(* Logix 5000 project; controller SX_V040001_C001 vendor 1 type 14 code 77 rev 16.22; software revision 16.04; part 26 of 35 *)
(* tags used below, declared in another part *)
   ALL_KINDS : INT[90];
   METERING : INT[44];
   PARAMETER : INT[501];
(* MainProgram, continued *)

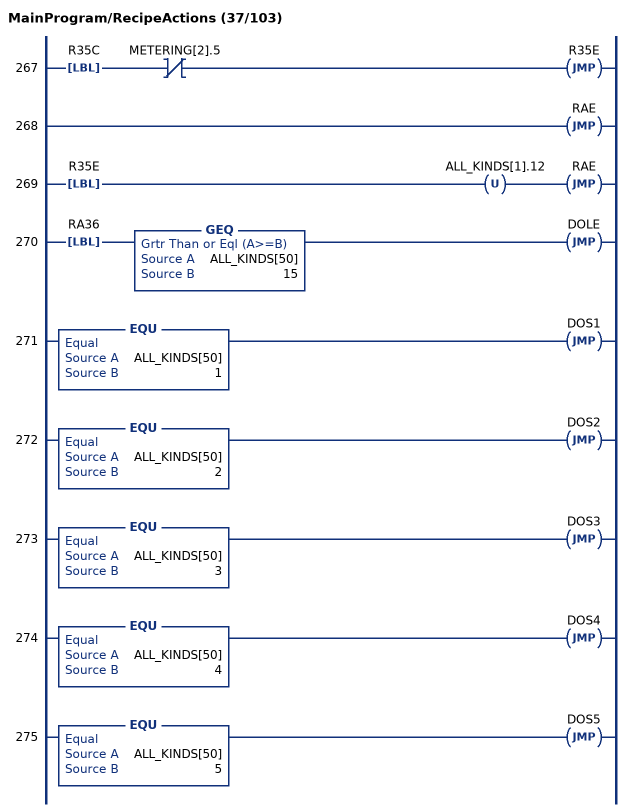
   [picture p568: MainProgram/RecipeActions rungs 267-275]
   267: LBL(R35C)XIO(METERING[2].5)JMP(R35E);
   268: JMP(RAE);
   269: LBL(R35E)OTU(ALL_KINDS[1].12)JMP(RAE);
   270: LBL(RA36)GEQ(ALL_KINDS[50],15)JMP(DOLE);
   271: EQU(ALL_KINDS[50],1)JMP(DOS1);
   272: EQU(ALL_KINDS[50],2)JMP(DOS2);
   273: EQU(ALL_KINDS[50],3)JMP(DOS3);
   274: EQU(ALL_KINDS[50],4)JMP(DOS4);
   275: EQU(ALL_KINDS[50],5)JMP(DOS5);
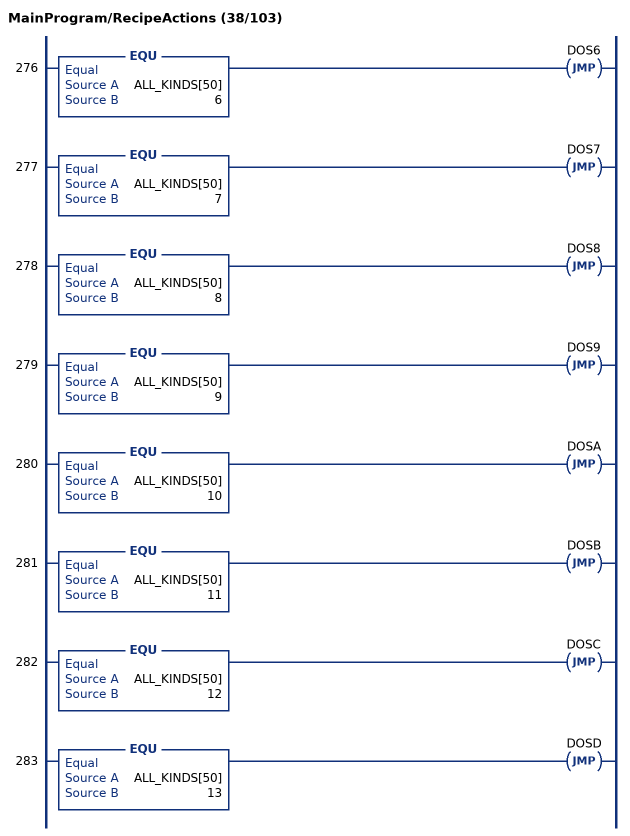
   276: EQU(ALL_KINDS[50],6)JMP(DOS6);
   277: EQU(ALL_KINDS[50],7)JMP(DOS7);
   278: EQU(ALL_KINDS[50],8)JMP(DOS8);
   279: EQU(ALL_KINDS[50],9)JMP(DOS9);
   280: EQU(ALL_KINDS[50],10)JMP(DOSA);
   281: EQU(ALL_KINDS[50],11)JMP(DOSB);
   282: EQU(ALL_KINDS[50],12)JMP(DOSC);
   283: EQU(ALL_KINDS[50],13)JMP(DOSD);
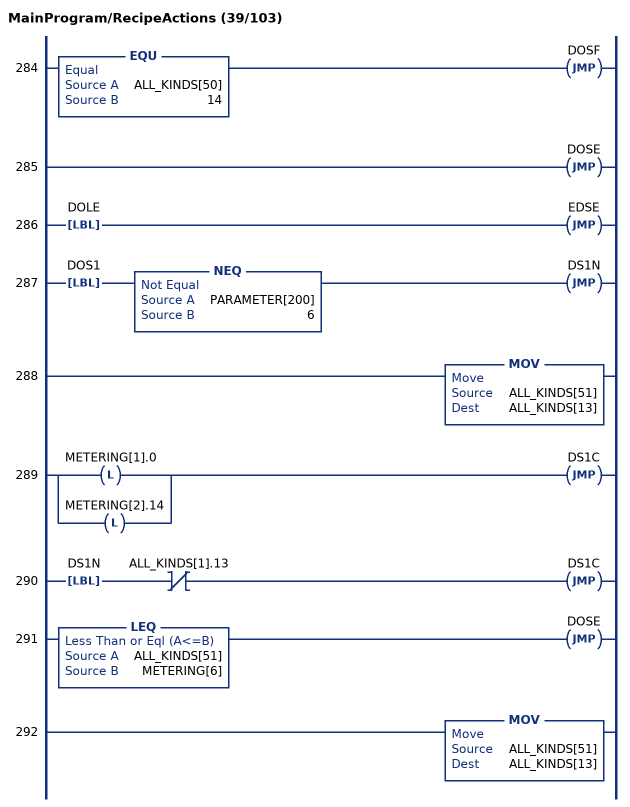
   284: EQU(ALL_KINDS[50],14)JMP(DOSF);
   285: JMP(DOSE);
   286: LBL(DOLE)JMP(EDSE);
   287: LBL(DOS1)NEQ(PARAMETER[200],6)JMP(DS1N);
   288: MOV(ALL_KINDS[51],ALL_KINDS[13]);
   289: [OTL(METERING[1].0) ,OTL(METERING[2].14) ]JMP(DS1C);
   290: LBL(DS1N)XIO(ALL_KINDS[1].13)JMP(DS1C);
   291: LEQ(ALL_KINDS[51],METERING[6])JMP(DOSE);
   292: MOV(ALL_KINDS[51],ALL_KINDS[13]);
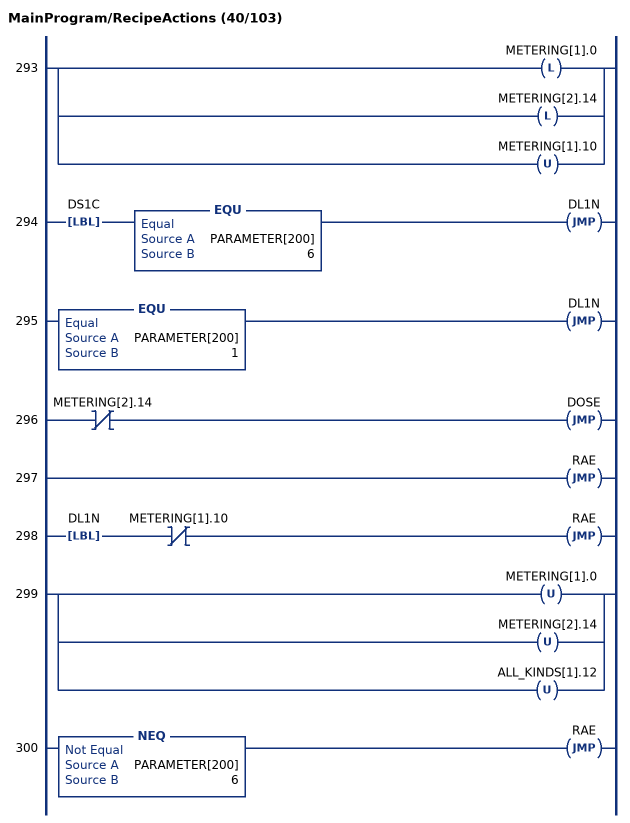
   293: [OTL(METERING[1].0) ,OTL(METERING[2].14) ,OTU(METERING[1].10) ];
   294: LBL(DS1C)EQU(PARAMETER[200],6)JMP(DL1N);
   295: EQU(PARAMETER[200],1)JMP(DL1N);
   296: XIO(METERING[2].14)JMP(DOSE);
   297: JMP(RAE);
   298: LBL(DL1N)XIO(METERING[1].10)JMP(RAE);
   299: [OTU(METERING[1].0) ,OTU(METERING[2].14) ,OTU(ALL_KINDS[1].12) ];
   300: NEQ(PARAMETER[200],6)JMP(RAE);
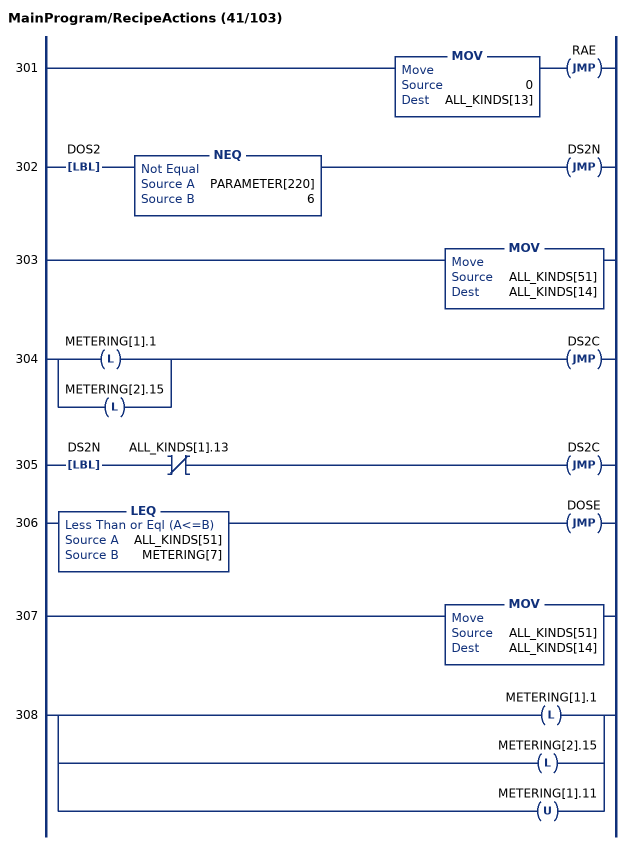
   301: MOV(0,ALL_KINDS[13])JMP(RAE);
   302: LBL(DOS2)NEQ(PARAMETER[220],6)JMP(DS2N);
   303: MOV(ALL_KINDS[51],ALL_KINDS[14]);
   304: [OTL(METERING[1].1) ,OTL(METERING[2].15) ]JMP(DS2C);
   305: LBL(DS2N)XIO(ALL_KINDS[1].13)JMP(DS2C);
   306: LEQ(ALL_KINDS[51],METERING[7])JMP(DOSE);
   307: MOV(ALL_KINDS[51],ALL_KINDS[14]);
   308: [OTL(METERING[1].1) ,OTL(METERING[2].15) ,OTU(METERING[1].11) ];
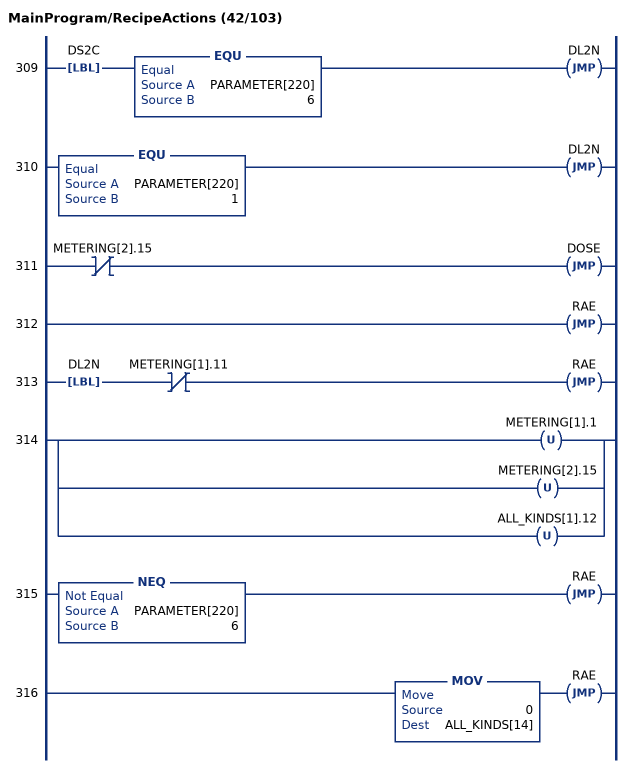
   309: LBL(DS2C)EQU(PARAMETER[220],6)JMP(DL2N);
   310: EQU(PARAMETER[220],1)JMP(DL2N);
   311: XIO(METERING[2].15)JMP(DOSE);
   312: JMP(RAE);
   313: LBL(DL2N)XIO(METERING[1].11)JMP(RAE);
   314: [OTU(METERING[1].1) ,OTU(METERING[2].15) ,OTU(ALL_KINDS[1].12) ];
   315: NEQ(PARAMETER[220],6)JMP(RAE);
   316: MOV(0,ALL_KINDS[14])JMP(RAE);
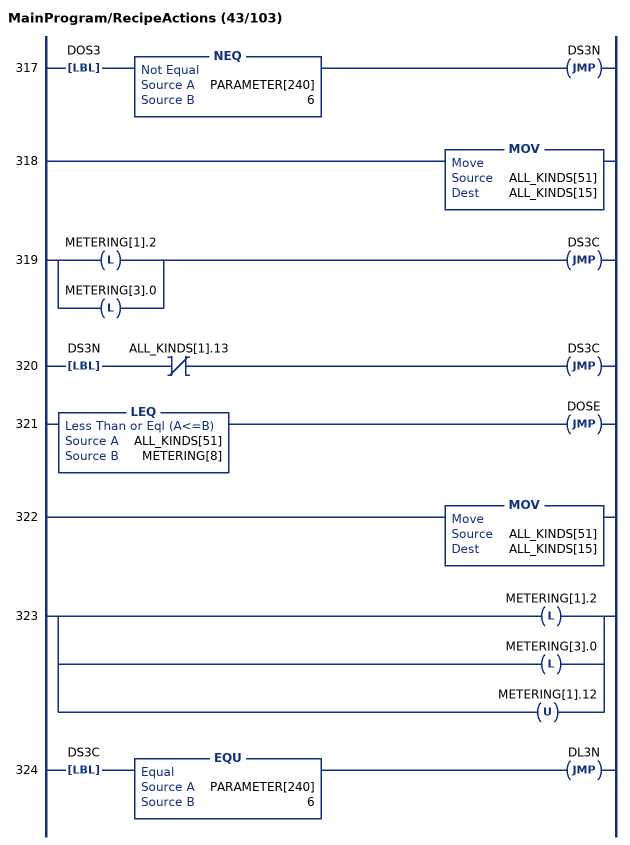
   317: LBL(DOS3)NEQ(PARAMETER[240],6)JMP(DS3N);
   318: MOV(ALL_KINDS[51],ALL_KINDS[15]);
   319: [OTL(METERING[1].2) ,OTL(METERING[3].0) ]JMP(DS3C);
   320: LBL(DS3N)XIO(ALL_KINDS[1].13)JMP(DS3C);
   321: LEQ(ALL_KINDS[51],METERING[8])JMP(DOSE);
   322: MOV(ALL_KINDS[51],ALL_KINDS[15]);
   323: [OTL(METERING[1].2) ,OTL(METERING[3].0) ,OTU(METERING[1].12) ];
   324: LBL(DS3C)EQU(PARAMETER[240],6)JMP(DL3N);
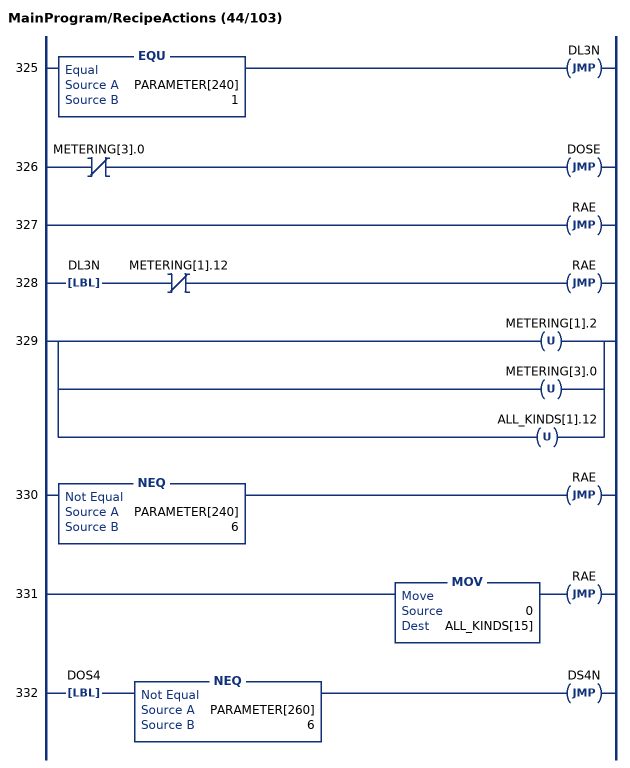
   325: EQU(PARAMETER[240],1)JMP(DL3N);
   326: XIO(METERING[3].0)JMP(DOSE);
   327: JMP(RAE);
   328: LBL(DL3N)XIO(METERING[1].12)JMP(RAE);
   329: [OTU(METERING[1].2) ,OTU(METERING[3].0) ,OTU(ALL_KINDS[1].12) ];
   330: NEQ(PARAMETER[240],6)JMP(RAE);
   331: MOV(0,ALL_KINDS[15])JMP(RAE);
   332: LBL(DOS4)NEQ(PARAMETER[260],6)JMP(DS4N);
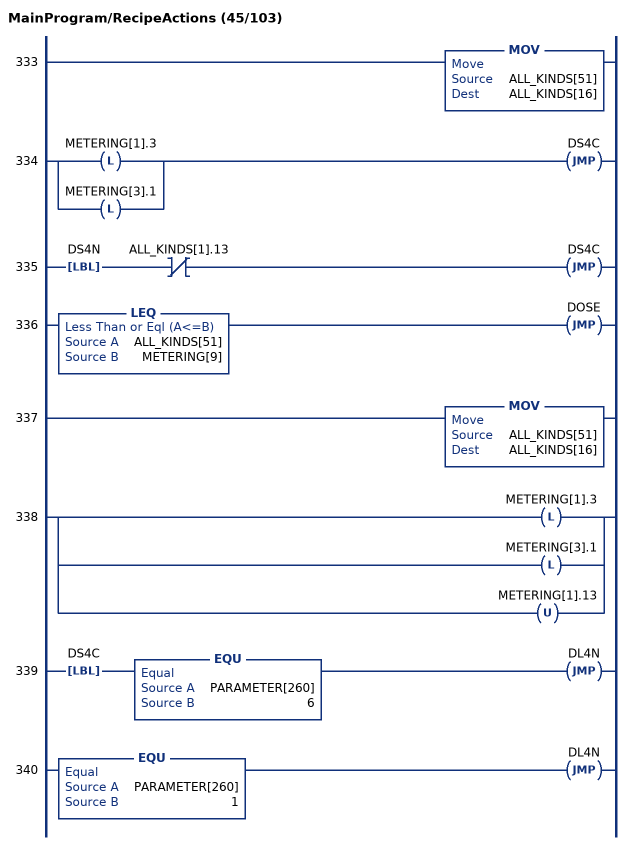
   333: MOV(ALL_KINDS[51],ALL_KINDS[16]);
   334: [OTL(METERING[1].3) ,OTL(METERING[3].1) ]JMP(DS4C);
   335: LBL(DS4N)XIO(ALL_KINDS[1].13)JMP(DS4C);
   336: LEQ(ALL_KINDS[51],METERING[9])JMP(DOSE);
   337: MOV(ALL_KINDS[51],ALL_KINDS[16]);
   338: [OTL(METERING[1].3) ,OTL(METERING[3].1) ,OTU(METERING[1].13) ];
   339: LBL(DS4C)EQU(PARAMETER[260],6)JMP(DL4N);
   340: EQU(PARAMETER[260],1)JMP(DL4N);
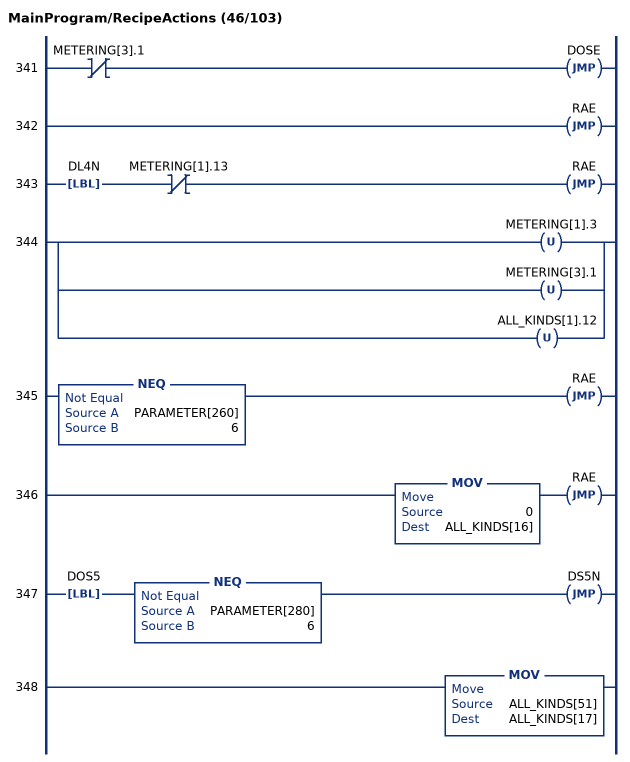
   341: XIO(METERING[3].1)JMP(DOSE);
   342: JMP(RAE);
   343: LBL(DL4N)XIO(METERING[1].13)JMP(RAE);
   344: [OTU(METERING[1].3) ,OTU(METERING[3].1) ,OTU(ALL_KINDS[1].12) ];
   345: NEQ(PARAMETER[260],6)JMP(RAE);
   346: MOV(0,ALL_KINDS[16])JMP(RAE);
   347: LBL(DOS5)NEQ(PARAMETER[280],6)JMP(DS5N);
   348: MOV(ALL_KINDS[51],ALL_KINDS[17]);
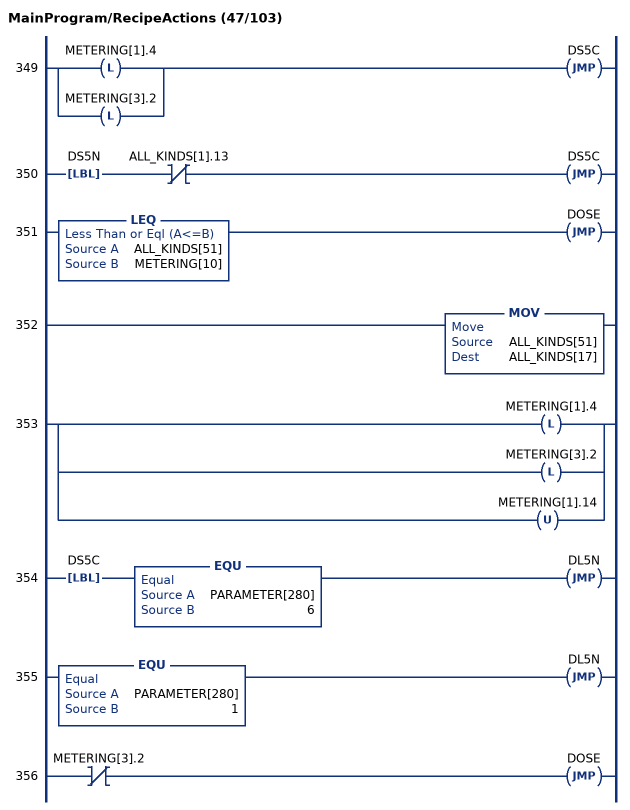
   349: [OTL(METERING[1].4) ,OTL(METERING[3].2) ]JMP(DS5C);
   350: LBL(DS5N)XIO(ALL_KINDS[1].13)JMP(DS5C);
   351: LEQ(ALL_KINDS[51],METERING[10])JMP(DOSE);
   352: MOV(ALL_KINDS[51],ALL_KINDS[17]);
   353: [OTL(METERING[1].4) ,OTL(METERING[3].2) ,OTU(METERING[1].14) ];
   354: LBL(DS5C)EQU(PARAMETER[280],6)JMP(DL5N);
   355: EQU(PARAMETER[280],1)JMP(DL5N);
   356: XIO(METERING[3].2)JMP(DOSE);
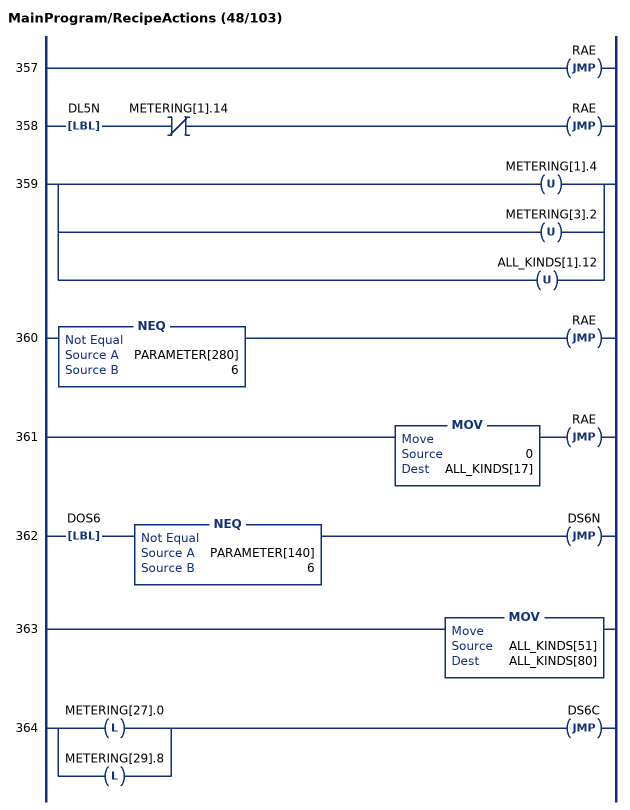
   357: JMP(RAE);
   358: LBL(DL5N)XIO(METERING[1].14)JMP(RAE);
   359: [OTU(METERING[1].4) ,OTU(METERING[3].2) ,OTU(ALL_KINDS[1].12) ];
   360: NEQ(PARAMETER[280],6)JMP(RAE);
   361: MOV(0,ALL_KINDS[17])JMP(RAE);
   362: LBL(DOS6)NEQ(PARAMETER[140],6)JMP(DS6N);
   363: MOV(ALL_KINDS[51],ALL_KINDS[80]);
   364: [OTL(METERING[27].0) ,OTL(METERING[29].8) ]JMP(DS6C);
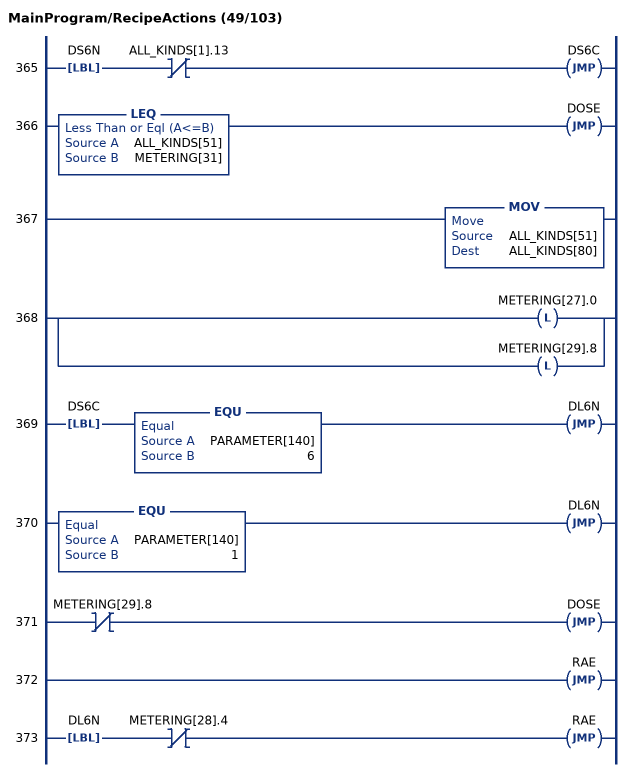
   365: LBL(DS6N)XIO(ALL_KINDS[1].13)JMP(DS6C);
   366: LEQ(ALL_KINDS[51],METERING[31])JMP(DOSE);
   367: MOV(ALL_KINDS[51],ALL_KINDS[80]);
   368: [OTL(METERING[27].0) ,OTL(METERING[29].8) ];
   369: LBL(DS6C)EQU(PARAMETER[140],6)JMP(DL6N);
   370: EQU(PARAMETER[140],1)JMP(DL6N);
   371: XIO(METERING[29].8)JMP(DOSE);
   372: JMP(RAE);
   373: LBL(DL6N)XIO(METERING[28].4)JMP(RAE);
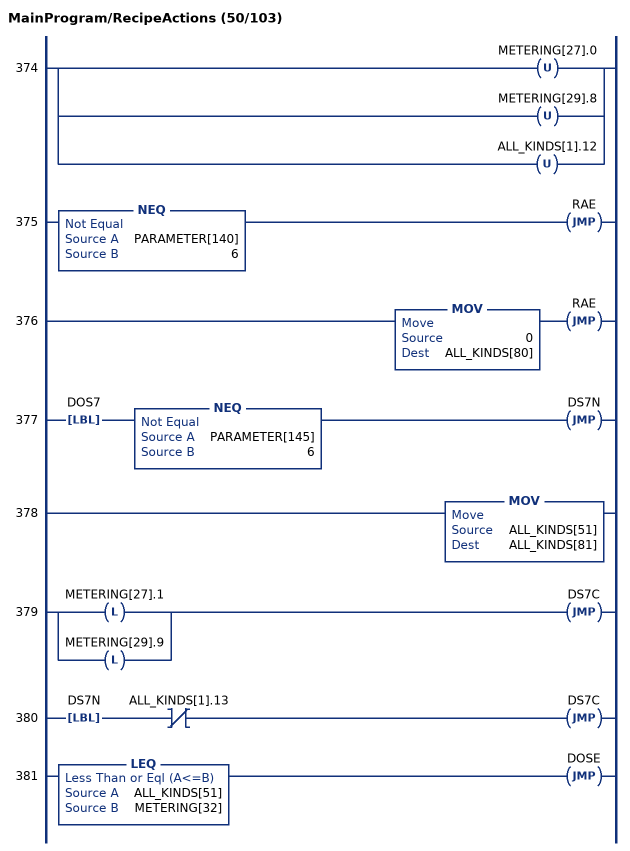
   374: [OTU(METERING[27].0) ,OTU(METERING[29].8) ,OTU(ALL_KINDS[1].12) ];
   375: NEQ(PARAMETER[140],6)JMP(RAE);
   376: MOV(0,ALL_KINDS[80])JMP(RAE);
   377: LBL(DOS7)NEQ(PARAMETER[145],6)JMP(DS7N);
   378: MOV(ALL_KINDS[51],ALL_KINDS[81]);
   379: [OTL(METERING[27].1) ,OTL(METERING[29].9) ]JMP(DS7C);
   380: LBL(DS7N)XIO(ALL_KINDS[1].13)JMP(DS7C);
   381: LEQ(ALL_KINDS[51],METERING[32])JMP(DOSE);
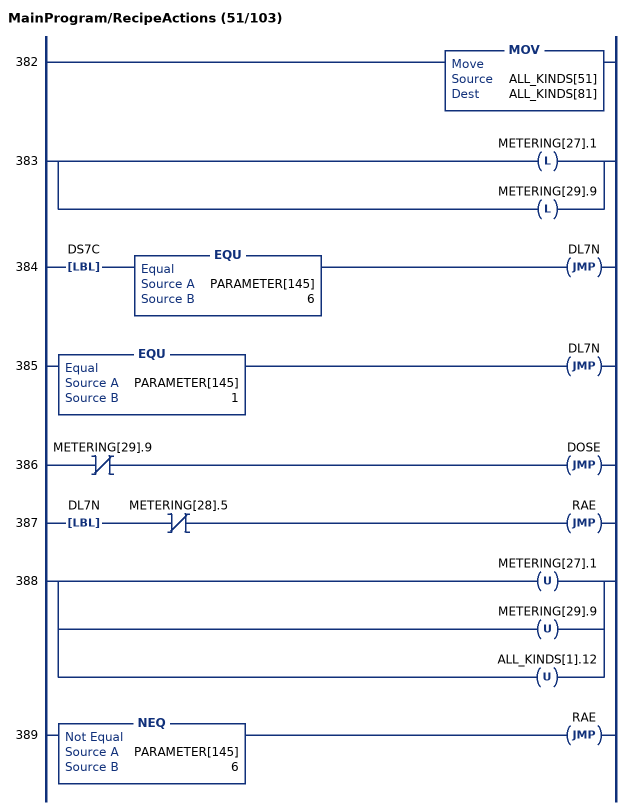
   382: MOV(ALL_KINDS[51],ALL_KINDS[81]);
   383: [OTL(METERING[27].1) ,OTL(METERING[29].9) ];
   384: LBL(DS7C)EQU(PARAMETER[145],6)JMP(DL7N);
   385: EQU(PARAMETER[145],1)JMP(DL7N);
   386: XIO(METERING[29].9)JMP(DOSE);
   387: LBL(DL7N)XIO(METERING[28].5)JMP(RAE);
   388: [OTU(METERING[27].1) ,OTU(METERING[29].9) ,OTU(ALL_KINDS[1].12) ];
   389: NEQ(PARAMETER[145],6)JMP(RAE);
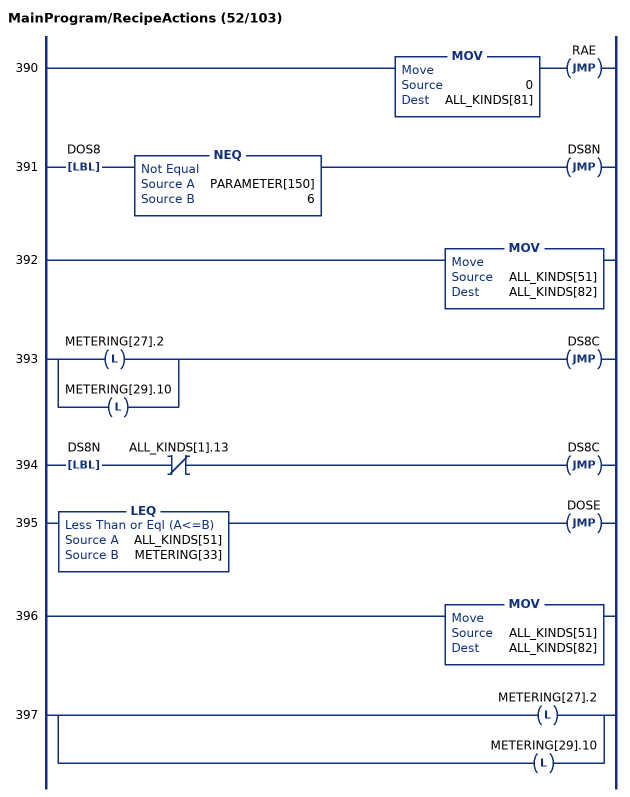
   390: MOV(0,ALL_KINDS[81])JMP(RAE);
   391: LBL(DOS8)NEQ(PARAMETER[150],6)JMP(DS8N);
   392: MOV(ALL_KINDS[51],ALL_KINDS[82]);
   393: [OTL(METERING[27].2) ,OTL(METERING[29].10) ]JMP(DS8C);
   394: LBL(DS8N)XIO(ALL_KINDS[1].13)JMP(DS8C);
   395: LEQ(ALL_KINDS[51],METERING[33])JMP(DOSE);
   396: MOV(ALL_KINDS[51],ALL_KINDS[82]);
   397: [OTL(METERING[27].2) ,OTL(METERING[29].10) ];
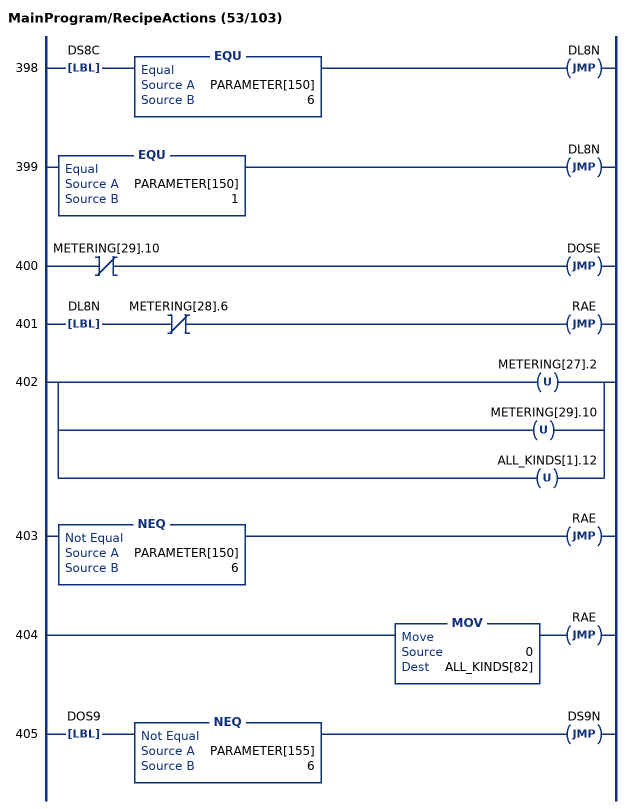
   398: LBL(DS8C)EQU(PARAMETER[150],6)JMP(DL8N);
   399: EQU(PARAMETER[150],1)JMP(DL8N);
   400: XIO(METERING[29].10)JMP(DOSE);
   401: LBL(DL8N)XIO(METERING[28].6)JMP(RAE);
   402: [OTU(METERING[27].2) ,OTU(METERING[29].10) ,OTU(ALL_KINDS[1].12) ];
   403: NEQ(PARAMETER[150],6)JMP(RAE);
   404: MOV(0,ALL_KINDS[82])JMP(RAE);
   405: LBL(DOS9)NEQ(PARAMETER[155],6)JMP(DS9N);
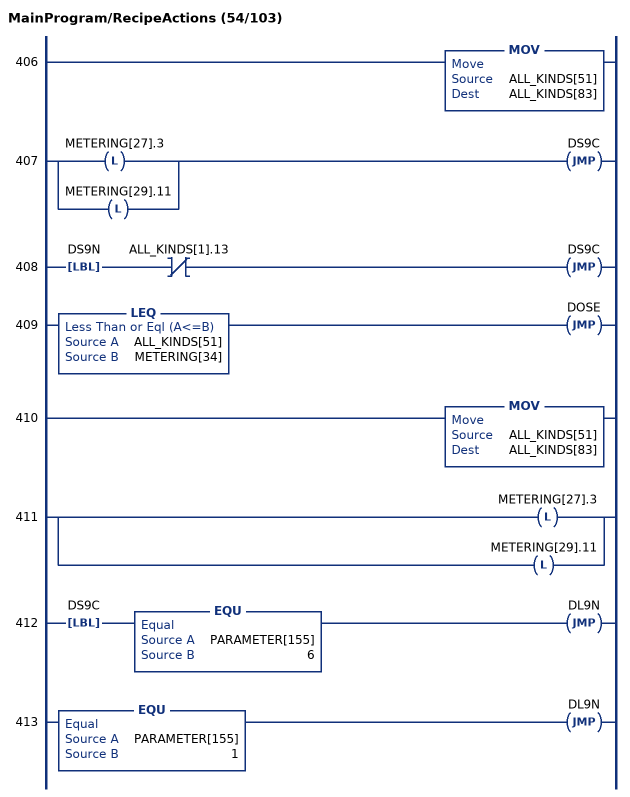
   406: MOV(ALL_KINDS[51],ALL_KINDS[83]);
   407: [OTL(METERING[27].3) ,OTL(METERING[29].11) ]JMP(DS9C);
   408: LBL(DS9N)XIO(ALL_KINDS[1].13)JMP(DS9C);
   409: LEQ(ALL_KINDS[51],METERING[34])JMP(DOSE);
   410: MOV(ALL_KINDS[51],ALL_KINDS[83]);
   411: [OTL(METERING[27].3) ,OTL(METERING[29].11) ];
   412: LBL(DS9C)EQU(PARAMETER[155],6)JMP(DL9N);
   413: EQU(PARAMETER[155],1)JMP(DL9N);
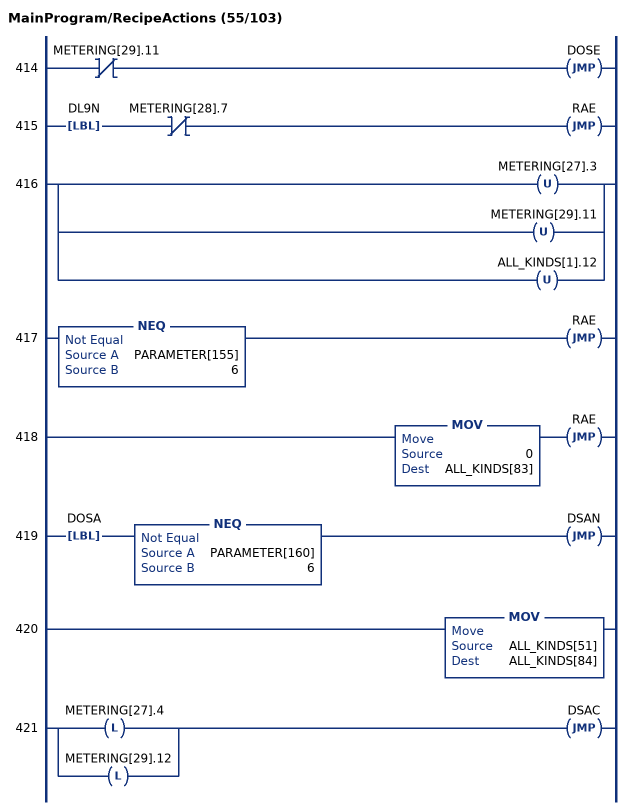
   414: XIO(METERING[29].11)JMP(DOSE);
   415: LBL(DL9N)XIO(METERING[28].7)JMP(RAE);
   416: [OTU(METERING[27].3) ,OTU(METERING[29].11) ,OTU(ALL_KINDS[1].12) ];
   417: NEQ(PARAMETER[155],6)JMP(RAE);
   418: MOV(0,ALL_KINDS[83])JMP(RAE);
   419: LBL(DOSA)NEQ(PARAMETER[160],6)JMP(DSAN);
   420: MOV(ALL_KINDS[51],ALL_KINDS[84]);
   421: [OTL(METERING[27].4) ,OTL(METERING[29].12) ]JMP(DSAC);
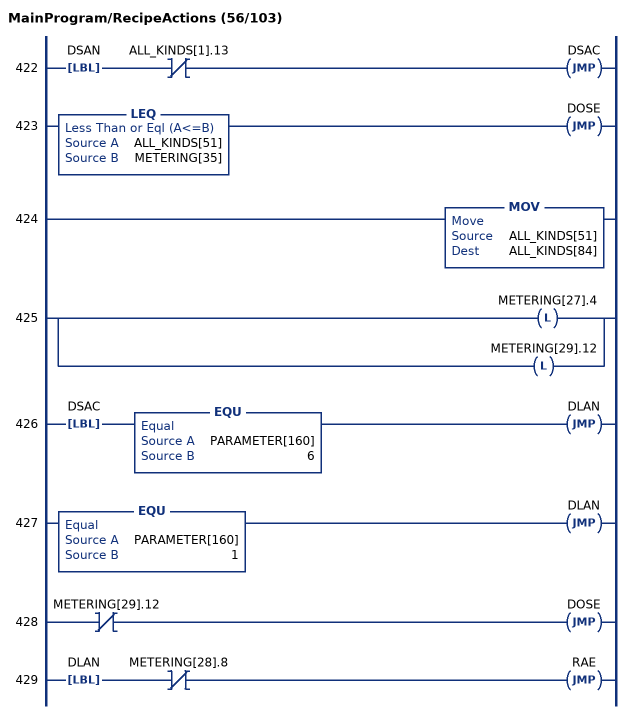
   422: LBL(DSAN)XIO(ALL_KINDS[1].13)JMP(DSAC);
   423: LEQ(ALL_KINDS[51],METERING[35])JMP(DOSE);
   424: MOV(ALL_KINDS[51],ALL_KINDS[84]);
   425: [OTL(METERING[27].4) ,OTL(METERING[29].12) ];
   426: LBL(DSAC)EQU(PARAMETER[160],6)JMP(DLAN);
   427: EQU(PARAMETER[160],1)JMP(DLAN);
   428: XIO(METERING[29].12)JMP(DOSE);
   429: LBL(DLAN)XIO(METERING[28].8)JMP(RAE);
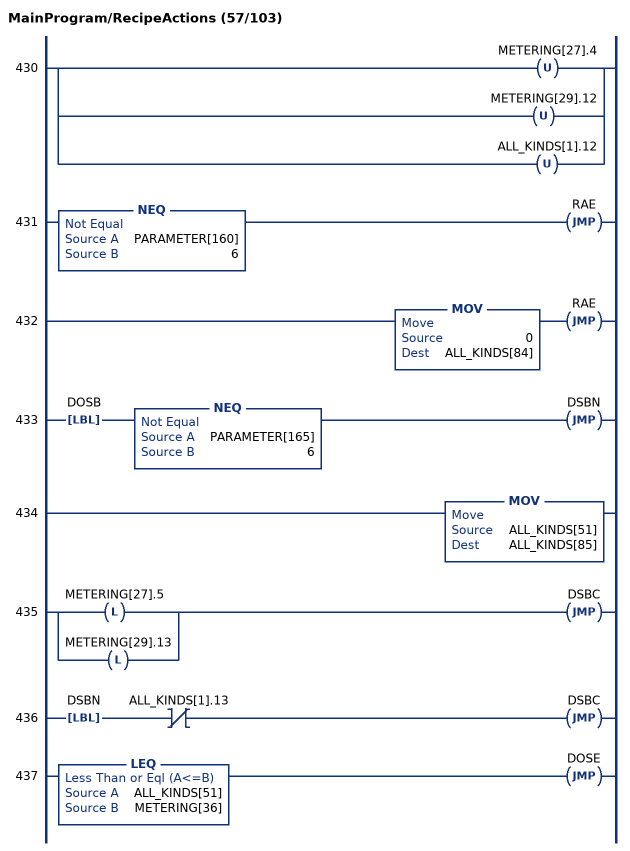
   430: [OTU(METERING[27].4) ,OTU(METERING[29].12) ,OTU(ALL_KINDS[1].12) ];
   431: NEQ(PARAMETER[160],6)JMP(RAE);
   432: MOV(0,ALL_KINDS[84])JMP(RAE);
   433: LBL(DOSB)NEQ(PARAMETER[165],6)JMP(DSBN);
   434: MOV(ALL_KINDS[51],ALL_KINDS[85]);
   435: [OTL(METERING[27].5) ,OTL(METERING[29].13) ]JMP(DSBC);
   436: LBL(DSBN)XIO(ALL_KINDS[1].13)JMP(DSBC);
   437: LEQ(ALL_KINDS[51],METERING[36])JMP(DOSE);
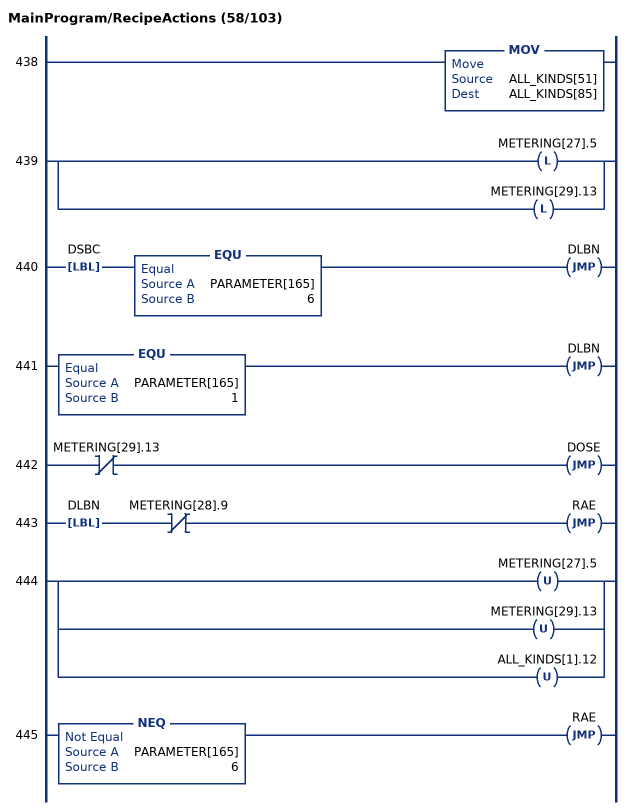
   438: MOV(ALL_KINDS[51],ALL_KINDS[85]);
   439: [OTL(METERING[27].5) ,OTL(METERING[29].13) ];
   440: LBL(DSBC)EQU(PARAMETER[165],6)JMP(DLBN);
   441: EQU(PARAMETER[165],1)JMP(DLBN);
   442: XIO(METERING[29].13)JMP(DOSE);
   443: LBL(DLBN)XIO(METERING[28].9)JMP(RAE);
   444: [OTU(METERING[27].5) ,OTU(METERING[29].13) ,OTU(ALL_KINDS[1].12) ];
   445: NEQ(PARAMETER[165],6)JMP(RAE);
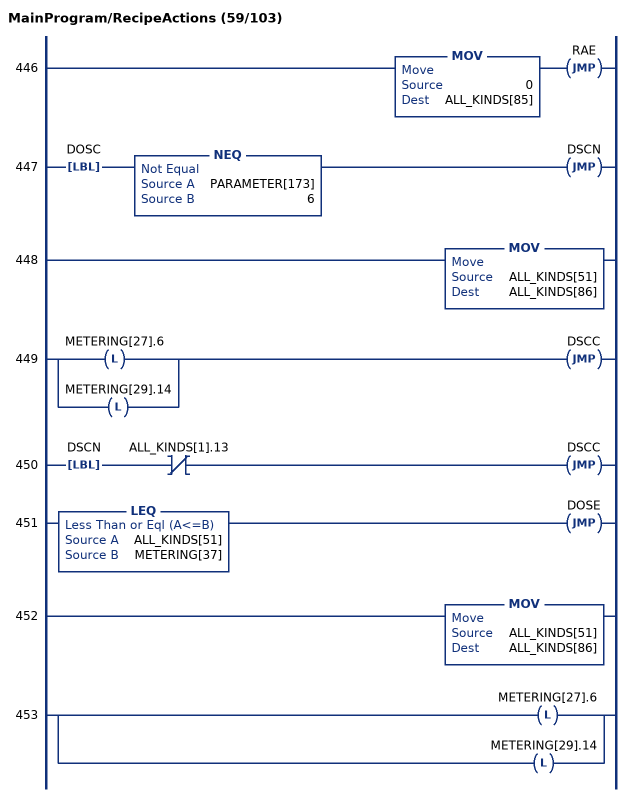
   446: MOV(0,ALL_KINDS[85])JMP(RAE);
   447: LBL(DOSC)NEQ(PARAMETER[173],6)JMP(DSCN);
   448: MOV(ALL_KINDS[51],ALL_KINDS[86]);
   449: [OTL(METERING[27].6) ,OTL(METERING[29].14) ]JMP(DSCC);
   450: LBL(DSCN)XIO(ALL_KINDS[1].13)JMP(DSCC);
   451: LEQ(ALL_KINDS[51],METERING[37])JMP(DOSE);
   452: MOV(ALL_KINDS[51],ALL_KINDS[86]);
   453: [OTL(METERING[27].6) ,OTL(METERING[29].14) ];
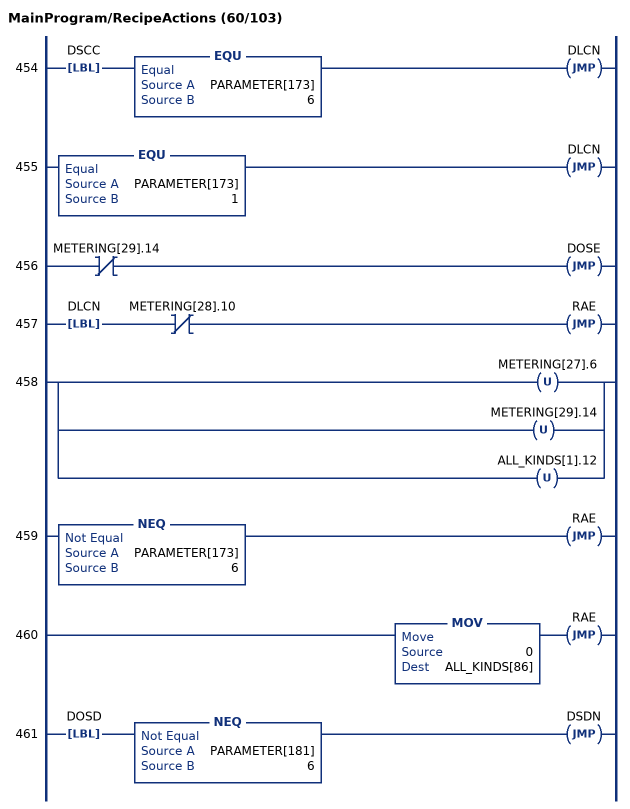
   454: LBL(DSCC)EQU(PARAMETER[173],6)JMP(DLCN);
   455: EQU(PARAMETER[173],1)JMP(DLCN);
   456: XIO(METERING[29].14)JMP(DOSE);
   457: LBL(DLCN)XIO(METERING[28].10)JMP(RAE);
   458: [OTU(METERING[27].6) ,OTU(METERING[29].14) ,OTU(ALL_KINDS[1].12) ];
   459: NEQ(PARAMETER[173],6)JMP(RAE);
   460: MOV(0,ALL_KINDS[86])JMP(RAE);
   461: LBL(DOSD)NEQ(PARAMETER[181],6)JMP(DSDN);
